Fanuc KAREL source: CA0044.KL

PROGRAM CA0044
%STACKSIZE=65535
%PRIORITY=65535
%NOLOCKGROUP
VAR
G : INTEGER
I : INTEGER
R : REAL
B : BOOLEAN
S : STRING[16]
AI : ARRAY[2] OF INTEGER
AR : ARRAY[2] OF REAL
P : XYZWPR
-- UNRESOLVED DECLARATIONS (source type spelling not recovered)
-- ST : TYPE_0x1100 (type_u16=0x1100)
-- V : TYPE_0x0013 (type_u16=0x0013)
ROUTINE F(P1 : INTEGER; P2 : INTEGER; P3 : INTEGER; P4 : INTEGER; P5 : INTEGER; P6 : INTEGER; P7 : INTEGER; P8 : INTEGER; P9 : INTEGER; P10 : INTEGER; P11 : INTEGER; P12 : INTEGER; P13 : INTEGER; P14 : INTEGER; P15 : INTEGER; P16 : INTEGER;
P17 : INTEGER; P18 : INTEGER; P19 : INTEGER; P20 : INTEGER; P21 : INTEGER; P22 : INTEGER; P23 : INTEGER; P24 : INTEGER) FROM CA0044
ROUTINE F
BEGIN
G=(G + 1)
END F
BEGIN
G=0
I=1
R=2.5
B=TRUE
S='A'
AI[1]=3
AR[1]=4.5
ST.A=5
ST.B=1087373312
-- UNSAFE_SOURCE_IR line 56: F(ARG_1_UNRESOLVED, ARG_2_UNRESOLVED, ARG_3_UNRESOLVED, ARG_4_UNRESOLVED, ARG_5_UNRESOLVED, ARG_6_UNRESOLVED, ARG_7_UNRESOLVED, ARG_8_UNRESOLVED, ARG_9_UNRESOLVED, ARG_10_UNRESOLVED, ARG_11_UNRESOLVED,
END CA0044
